Omron CX-Programmer project NewProject (CX-Programmer 9.73)

# PLC NewPLC1: CP1E N30

## Global symbols (name address type ; comment)
0.00 BOOL  ; sw1
100.00 BOOL  ; G1
100.01 BOOL  ; G2
100.02 BOOL  ; G3
100.03 BOOL  ; G4
1.03 BOOL  ; Stop

## Program NewProgram1 (cyclic task 0)

### Section Section1

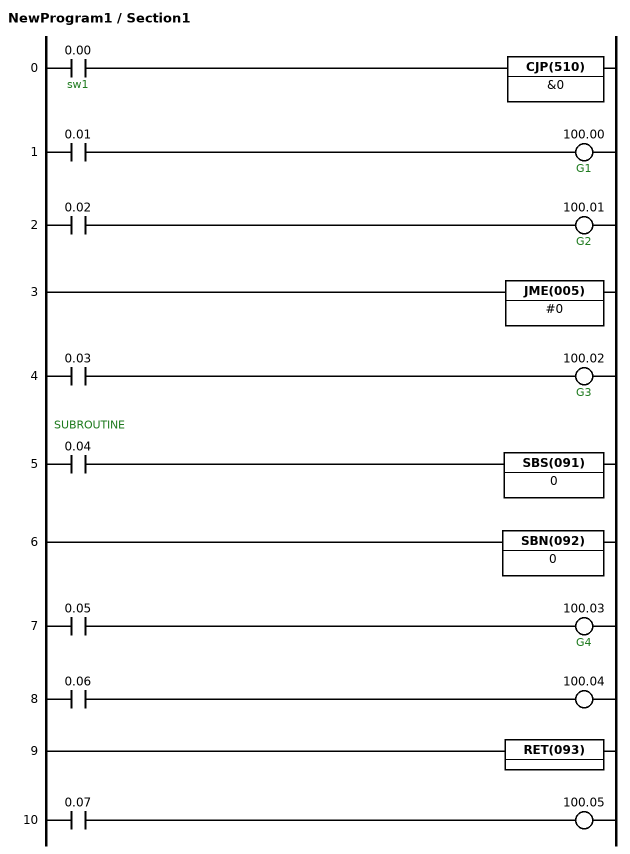
; rung 0
LD 0.00  ; sw1
CJP(510) &0
; rung 1
LD 0.01
OUT 100.00  ; G1
; rung 2
LD 0.02
OUT 100.01  ; G2
; rung 3
JME(005) #0
; rung 4
LD 0.03
OUT 100.02  ; G3
; rung 5: SUBROUTINE
LD 0.04
SBS(091) 0
; rung 6
SBN(092) 0
; rung 7
LD 0.05
OUT 100.03  ; G4
; rung 8
LD 0.06
OUT 100.04
; rung 9
RET(093)
; rung 10
LD 0.07
OUT 100.05

### Section filled_process

### Section END
; rung 0
END(001)